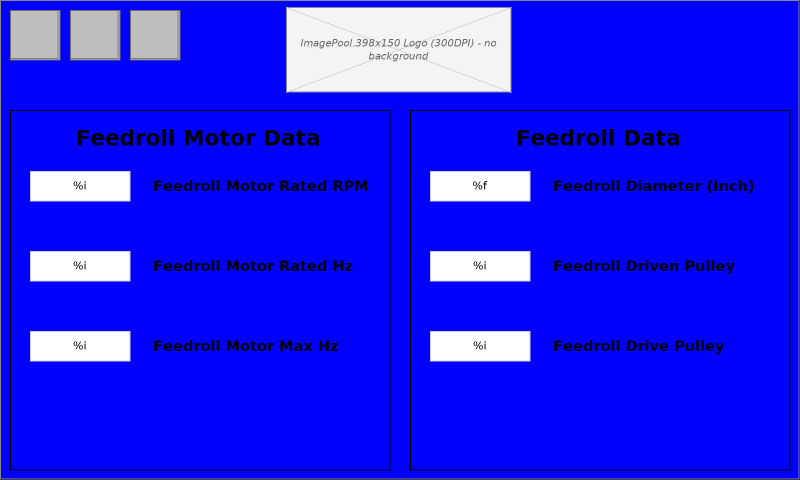
VISUALIZATION Feedroll_Settings  // 800x480
    Rectangle (0,0 800x480)
    Rectangle (10,110 380x360)
    Textfield (30,171 100x30), "%i", text variable: GVL.FeedrollMot_Rated_RPM
        OnMouseClick: write the text variable via VisuDialogs.Numpad
    Rectangle (410,110 380x360)
    Textfield (30,251 100x30), "%i", text variable: GVL.FeedrollMot_Rated_Hz
        OnMouseClick: write the text variable via VisuDialogs.Numpad
    Textfield (30,331 100x30), "%i", text variable: GVL.FeedrollMot_Max_Hz
        OnMouseClick: write the text variable via VisuDialogs.Numpad
    Image (286,7 225x85), image: ImagePool.398x150 Logo (300DPI) - no background
        OnMouseClick: change screen: Home
    Button (70,10 50x50), image: VisuSymbols.Symbols.Home
        OnMouseClick: change screen: Home
    Label (20,120 357x36), "Feedroll Motor Data"
    Label (420,120 357x36), "Feedroll Data"
    Button (10,10 50x50), image: VisuSymbols.Symbols.TriangleLeft
        OnMouseClick: change screen: Previous Home
    Textfield (430,171 100x30), "%f", text variable: GVL.Feedroll_Diameter_Inch
        OnMouseClick: write the text variable via VisuDialogs.Numpad
    Textfield (430,251 100x30), "%i", text variable: GVL.Feedroll_Driven_Pulley
        OnMouseClick: write the text variable via VisuDialogs.Numpad
    Textfield (430,331 100x30), "%i", text variable: GVL.Feedroll_Drive_Pulley
        OnMouseClick: write the text variable via VisuDialogs.Numpad
    Label (150,171 225x30), "Feedroll Motor Rated RPM"
    Label (150,251 225x30), "Feedroll Motor Rated Hz"
    Label (150,331 225x30), "Feedroll Motor Max Hz"
    Label (550,171 225x30), "Feedroll Diameter (Inch)"
    Label (550,251 225x30), "Feedroll Driven Pulley"
    Label (550,331 225x30), "Feedroll Drive Pulley"
    Button (130,10 50x50), image: VisuSymbols.Symbols.TwoWheels
        OnMouseClick: change screen: Settings_Menu
END_VISUALIZATION

(* stored: Version 1.1.0.1, ProductVersion 3.1.4024.12
   Visu Feedroll_Settings: Id {30eb8320-3e8a-4da7-8581-32db0ad18313} *)
